(* Schneider Machine Expert - Basic project Traffic timer changed, file version 1.9.0.0 *)
(* ProjectInformations: Name=New project *)

HARDWARE
  Cpu 0: TM221CE16R
  EthernetConfiguration: NetworkName=M221, IpAllocationMode=FixedAddress, IpAddress=0.0.0.0, SubnetMask=0.0.0.0
  SerialLineConfiguration: Baud=Baud19200, Parity=ParityEven, DataBits=DataBits8, StopBits=StopBits1, PhysicalMedium=PhysicalMediumRs485, TransmissionMode=TransmissionModeModbusRtu, SlaveId=1, Addressing=SlaveAddressing
  MastTask: UsePeriodScanMode=false, PeriodScan=100
  FastTask: Period=255
  CpuBehavior: StartingMode=StartAsPreviousState, AutoSaveRamOnEeprom=true, WatchdogPeriod=250

SYMBOLS  (address, symbol, comment, settings)
  %TM1        [Preset=5, Base=OneSecond]
  %TM2        [Preset=2, Base=OneSecond]
  %TM3        [Preset=5, Base=OneHundredMilliSeconds]
  %TM5        [Preset=3, Base=OneSecond]

POU New POU
  (* SectionNumber=1 *)

// Rung 0
  BLK %TM5
  LD %I0.0
  ANDN %M2
  IN
  OUT_BLK
  LD Q
  ST %M0
  END_BLK
  // as ST:
  //   %TM5(IN := %I0.0 AND NOT %M2);
  //   %M0 := %TM5.Q;

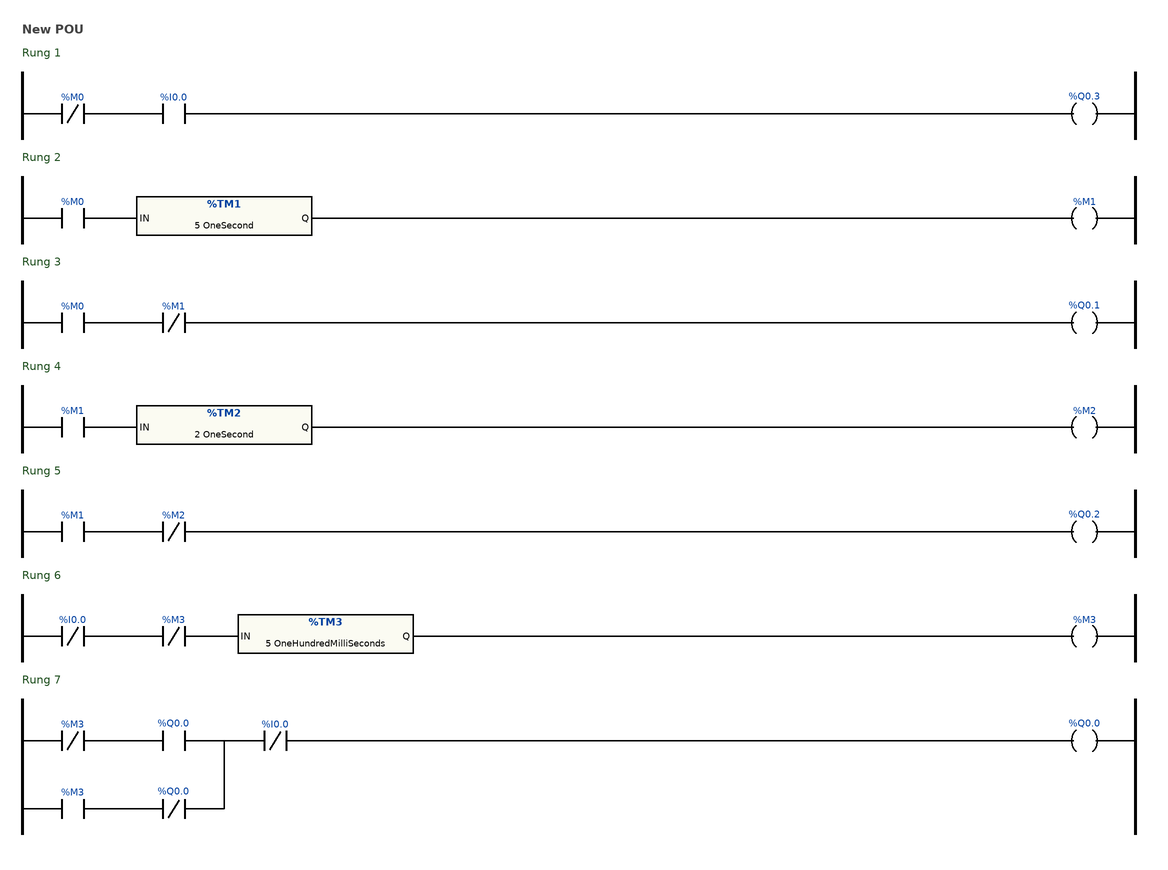

// Rung 1
  LDN %M0
  AND %I0.0
  ST %Q0.3
  // as ST:
  //   %Q0.3 := NOT %M0 AND %I0.0;

// Rung 2
  BLK %TM1
  LD %M0
  IN
  OUT_BLK
  LD Q
  ST %M1
  END_BLK
  // as ST:
  //   %TM1(IN := %M0);
  //   %M1 := %TM1.Q;

// Rung 3
  LD %M0
  ANDN %M1
  ST %Q0.1
  // as ST:
  //   %Q0.1 := %M0 AND NOT %M1;

// Rung 4
  BLK %TM2
  LD %M1
  IN
  OUT_BLK
  LD Q
  ST %M2
  END_BLK
  // as ST:
  //   %TM2(IN := %M1);
  //   %M2 := %TM2.Q;

// Rung 5
  LD %M1
  ANDN %M2
  ST %Q0.2
  // as ST:
  //   %Q0.2 := %M1 AND NOT %M2;

// Rung 6
  BLK %TM3
  LDN %I0.0
  ANDN %M3
  IN
  OUT_BLK
  LD Q
  ST %M3
  END_BLK
  // as ST:
  //   %TM3(IN := NOT %I0.0 AND NOT %M3);
  //   %M3 := %TM3.Q;

// Rung 7
  LDN %M3
  AND %Q0.0
  OR( %M3
  ANDN %Q0.0
  )
  ANDN %I0.0
  ST %Q0.0
  // as ST:
  //   %Q0.0 := (NOT %M3 AND %Q0.0 OR %M3 AND NOT %Q0.0) AND NOT %I0.0;
